FUNCTION_BLOCK T_BaseAlarms EXTENDS T_NamedBase
VAR
	alarms : ARRAY[E_BaseAlarms.InitReferenceEvent..E_BaseAlarms.InvalidInterface] OF FB_TcAlarm;
END_VAR
VAR CONSTANT
	USE_DEFAULT_TIMESTAMP : ULINT := 0; // If default then it will use system time, else it will use timestamp 
  //https://infosys.beckhoff.com/english.php?content=../content/1033/tc3_eventlogger/5050505739.html&id=8432917619912920197
END_VAR

PROPERTY AlarmsArray : REFERENCE TO ARRAY[E_BaseAlarms.InitReferenceEvent..E_BaseAlarms.InvalidInterface] OF FB_TcAlarm
GET
AlarmsArray REF= alarms;
END_GET
END_PROPERTY

METHOD ClearAlarmIfRaised
VAR_INPUT
	alarm : E_BaseAlarms;
	resetConfirmation : BOOL;
END_VAR
IF NOT alarms[alarm].bRaised THEN
	RETURN;
END_IF

alarms[alarm].Clear(USE_DEFAULT_TIMESTAMP,resetConfirmation);
END_METHOD

METHOD RaiseAlarmWithStringParameters
VAR_INPUT
	alarm : E_BaseAlarms;

	String_1 : STRING; //! First string parameter
	String_2 : STRING; //! Second string parameter
	String_3 : STRING; //! Third string parameter

END_VAR
IF alarms[alarm].bRaised THEN
	RETURN;
END_IF

alarms[alarm].ipArguments.Clear();
IF String_1 <> '' THEN
	alarms[alarm].ipArguments.AddString(String_1);
END_IF

IF String_2 <> '' THEN
	alarms[alarm].ipArguments.AddString(String_2);
END_IF

IF String_3 <> '' THEN
	alarms[alarm].ipArguments.AddString(String_3);
END_IF

alarms[alarm].Raise(USE_DEFAULT_TIMESTAMP);
END_METHOD

END_FUNCTION_BLOCK

(* stored: Version 1.1.0.1, ProductVersion 3.1.4024.12
   POU T_BaseAlarms: Id {72ce3e27-50a6-4915-a06e-f6359f7eaba7}, SpecialFunc None
   Property AlarmsArray: Id {cf72b990-38ce-4505-806f-9a0ca9dbd4f6}
   Get Get: Id {ae170d6e-5f63-4195-83b1-2bd963ae3754}
   Method ClearAlarmIfRaised: Id {cdcba135-bb29-4c73-a463-8ac949a9728a}
   Method RaiseAlarmWithStringParameters: Id {0f4d0e4c-859c-44b0-99f0-051c92c550d7} *)
